// TIA Portal V20 export
// export: Created 2025-12-01T14:57:43.2505605Z, ExportSetting None, DisplayName Totally Integrated Automation Portal, DisplayVersion V20 Update 3, DisplayName TIA Portal Openness, DisplayVersion V20 Update 3, DisplayName TIA Portal Version Control Interface, DisplayVersion V20 Update 3, DisplayName STEP 7 Professional, DisplayVersion V20 Update 3, DisplayName STEP 7 Safety, DisplayVersion V20 Update 2, DisplayName WinCC Basic/Comfort/Advanced, DisplayVersion V20 Update 3, DisplayName WinCC Professional, DisplayVersion V20 Update 3, DisplayName WinCC Unified, DisplayVersion V20 Update 3
FUNCTION_BLOCK "FB955_Leer_Ips_Gateways"   // FB955, LAD
{ S7_Optimized_Access := 'FALSE' }
// stored: AutoNumber false, SetENOAutomatically true
   VAR
      Gateway { S7_SetPoint := 'True'} : Array[1..16] of "LPNDR_ReadGlobalInfo";
      lee { S7_SetPoint := 'True'} : Array[1..16] of Bool;
   END_VAR
   VAR_TEMP
      i : Int;
   END_VAR
BEGIN

REGION Network 1 (SCL): LEER LOS NOMBRES Y LAS IPS DE TODOS LOS GATEWAYS QUE TENEMOS QUE DIAGNOSTICAR
   FOR #i := 1 TO 16  BY 1 DO
       IF (("DB1904_Datos_Config_Gateways".Gateway[#i].Diagnosticar=true)AND("DB1903_ASI_DIAG".IP_GW[#i].nameOfStation=''))THEN
           #lee[#i] := true;
           #Gateway[#i](execute :=((#lee[#i])AND(NOT (#Gateway[#i].done))),
                        hwId := "DB1904_Datos_Config_Gateways".Gateway[#i].hwld,done=>#Gateway[#i].done);

           IF #Gateway[#i].done = TRUE THEN
               "DB1903_ASI_DIAG".IP_GW[#i].ipAdress := #Gateway[#i].InterfaceInformation.ipAdress;
               "DB1903_ASI_DIAG".IP_GW[#i].nameOfStation := #Gateway[#i].InterfaceInformation.nameOfStation;
               #lee[#i] := false;
           END_IF;
   ELSIF ("DB1904_Datos_Config_Gateways".Gateway[#i].Diagnosticar=false) THEN
       "DB1903_ASI_DIAG".IP_GW[#i].ipAdress[0] := 0;
       "DB1903_ASI_DIAG".IP_GW[#i].ipAdress[1] := 0;
       "DB1903_ASI_DIAG".IP_GW[#i].ipAdress[2] := 0;
       "DB1903_ASI_DIAG".IP_GW[#i].ipAdress[3] := 0;
       "DB1903_ASI_DIAG".IP_GW[#i].nameOfStation := '';
       #Gateway[#i].InterfaceInformation.ipAdress[0] := 0;
       #Gateway[#i].InterfaceInformation.ipAdress[1] := 0;
       #Gateway[#i].InterfaceInformation.ipAdress[2] := 0;
       #Gateway[#i].InterfaceInformation.ipAdress[3] := 0;
       #Gateway[#i].InterfaceInformation.nameOfStation := '';
       #lee[#i] := false;

   END_IF;


   END_FOR;
END_REGION
END_FUNCTION_BLOCK
